PROGRAM P_Feeder
VAR
	bStartFeeder : BOOL;
	bFeederOK: BOOL;
	//dut_FeedingState : FeedingState;
	fbFb_FeedingStateCheck: Fb_FeedingStateCheck;	
//-----------------------------------Feeder Mode -------------------------//
	iFeederMode : INT;	
	bGoCounter, bSetCounter AT %Q*:BOOL;
	wFrequencyValue, wTargetCounterValue, wSetCounterValue AT %Q*:WORD;
	wCounterValue AT %I*:WORD;
	nState, nCntCycle:UDINT;
	bStart:BOOL;
	wFrequencyValue_Test:WORD:=200;
	nPrevValue			:WORD;
	wTargetCounterValue_Test:WORD:=180;
	bHitTop : BOOL;
	bHitBottom : BOOL;
	bTargetDistanceHitUP	: BOOL;
	bTargetDistanceHitDown	: BOOL;

//------------------------------------CASE-------------------------------//
	ifeedercase : INT;

(* For reference
	State_Init 					:= 1,
	State_AutoStart         	:= 2,
	State_AutoHysterisis    	:= 3,
	State_AutoStop          	:= 4,
	State_AutoTopSensorReached 	:= 5,
	State_AutoFinalPosition     := 6,
	State_AutoBackToInit        := 7,
	State_Feeding				:= 8,
	State_Override				:= 9,
	State_Error					:= 10,
	State_ManualMoveUp			:= 11,
	State_ManualMoveDown    	:= 12
*)	
//-------------------------Simulated Values-----------------------------//
nCurrentValue 	: DWORD;
nTargetValue	: DWORD;
	
END_VAR
VAR_INPUT
	bStartCommand : BOOL;
END_VAR

IF GVL.bHmiSimulation THEN
	GVL.stHMIsimul:=GVL.stHMI;
	iFeederMode:=FeederMode.Mode_Simulation;
END_IF 
IF NOT GVL.bHmiSimulation THEN
	GVL.stHMI:=GVL.stHMI;
	iFeederMode:=FeederMode.Mode_Standard;
END_IF

CASE ifeedercase OF

FeedingState.State_Init 			:	//Awaiting for command   
	IF GVL.stHMI.bAuto  THEN
		ifeedercase:=FeedingState.State_AutoStart;
	END_IF
	IF GVL.stHMI.bFeederManualDown THEN
		ifeedercase:=FeedingState.State_ManualMoveDown;	
	END_IF
	IF GVL.stHMI.bFeederManualUp THEN
		ifeedercase:=FeedingState.State_ManualMoveUp;
	END_IF	
	IF NOT (iFeederMode=FeederMode.Mode_Simulation) THEN // go back to init
		iFeederCase:=FeedingState.State_Init;
		wTargetCounterValue:=0;
		nPrevValue:=0;	
		bHitTop:=FALSE;	
		bHitBottom:=FALSE;
		bTargetDistanceHitUp:=FALSE;
		bTargetDistanceHitDown:=FALSE;
		nState:=0;
	END_IF
	
FeedingState.State_AutoStart            : 	//Start 

	IF NOT bStartFeeder THEN
		ifeedercase:= FeedingState.State_AutoBackToInit;
	END_IF
	IF GVL.bHmiSimulation THEN
		//Adding Feeder movement simulation
		;
	END_IF
FeedingState.State_AutoHysterisis       : 
FeedingState.State_AutoStop             : 
FeedingState.State_AutoTopSensorReached :	
FeedingState.State_AutoFinalPosition    : 
FeedingState.State_AutoBackToInit       : 
FeedingState.State_Feeding				:        
FeedingState.State_Override				:       
FeedingState.State_Error				:	
     
FeedingState.State_ManualMoveUp			:
	IF iFeederMode=FeederMode.Mode_Simulation THEN
		CASE nState OF
				0: //Check ongoing or Initial Start
					IF gvl.stHMI.bFeederManualUp THEN
						IF NOT (bHitTop OR bTargetDistanceHitUp) THEN
							IF nPrevValue=0 
							AND wTargetCounterValue=0 THEN // Coming from initialization
								nState:=20;
							END_IF
							IF wTargetCounterValue>nPrevValue THEN //Continuation
								nPrevValue:=wTargetCounterValue;
								nState:=20;
							END_IF
						ELSE
							nState:=0;
							nPrevValue:=wTargetCounterValue;
						END_IF
					END_IF	
					
				20://Increment and making sure previous values are recorded.			
							IF (wTargetCounterValue>nPrevValue) THEN
								nState:=30;
							END_IF
							IF (wTargetCounterValue=nPrevValue) THEN
								wTargetCounterValue:=wTargetCounterValue+1;
								nState:=20;
							END_IF

				30:	//Check if reached target or not
					IF wTargetCounterValue < wTargetCounterValue_Test THEN //not reached
						nstate:=0;
					END_IF
					IF wTargetCounterValue >= wTargetCounterValue_Test OR bHitTop THEN // Reached sensor top or movement set
						nState:=40;
					END_IF
				40:	
					nState:=0;
					bTargetDistanceHitUp:=TRUE;
					bFeederOK :=TRUE;
					
				
		END_CASE
	END_IF
	IF iFeederMode=FeederMode.Mode_Jog THEN
		;
	END_IF
	ifeedercase:= FeedingState.State_Init;
	
FeedingState.State_ManualMoveDown		:
	IF iFeederMode=FeederMode.Mode_Simulation THEN
		CASE nState OF
				0: //Check ongoing or Initial Start
					IF gvl.stHMI.bFeederManualDown THEN
						IF NOT (bHitBottom OR bTargetDistanceHitDown) THEN
							IF nPrevValue=0 
							AND wTargetCounterValue=0 THEN // Coming from initialization
								nState:=20;
							END_IF
							IF wTargetCounterValue>nPrevValue THEN //Continuation
								nPrevValue:=wTargetCounterValue;
								nState:=20;
							END_IF
						ELSE
							nState:=0;
							nPrevValue:=wTargetCounterValue;
						END_IF
					END_IF	
					
				20://Increment and making sure previous values are recorded.			
							IF (wTargetCounterValue>nPrevValue) THEN
								nState:=30;
							END_IF
							IF (wTargetCounterValue=nPrevValue) THEN
								wTargetCounterValue:=wTargetCounterValue+1;
								nState:=20;
							END_IF

				30:	//Check if reached target or not
					IF wTargetCounterValue < wTargetCounterValue_Test THEN //not reached
						nstate:=0;
					END_IF
					IF wTargetCounterValue >= wTargetCounterValue_Test OR bHitTop THEN // Reached sensor top or movement set
						nState:=40;
					END_IF
				40:	
					nState:=0;
					bTargetDistanceHitDown:=TRUE;
				
		END_CASE
	END_IF
	IF iFeederMode=FeederMode.Mode_Jog THEN
		;
	END_IF
	ifeedercase:= FeedingState.State_Init;
	

END_CASE

END_PROGRAM

(* stored: Version 1.1.0.1, ProductVersion 3.1.4024.12
   POU P_Feeder: Id {1b62ab0e-a2dc-4978-80be-8223d6880511}, SpecialFunc None *)
